(* CoDeSys 2.3 export: ST_ISSUE94_BYTE.EXP *)

(* Data type *)
TYPE ST_Issue94_Byte :
STRUCT
	ByteValue : BYTE;
END_STRUCT
END_TYPE
